FUNCTION_BLOCK FB_WriteRegsExample
VAR
	fbWriteRegisters : FB_MBWriteRegs;
	nWriteValueArray : ARRAY[0..9] OF INT;
	wWriteRegsValueConvertToWord : WORD;
	eWriteState : (WAIT, TRIGGER, WRITE);
	fbTriggerStart : R_TRIG;
	fbTriggerStop : R_TRIG;
	//cbLength: UINT;
	
END_VAR

fbTriggerStart();
IF fbTriggerStart.Q THEN
	IF eWriteState = WAIT THEN
		 eWriteState := TRIGGER;
	END_IF
END_IF
IF fbTriggerStop.CLK THEN
	fbWriteRegisters(bExecute := FALSE);
	eWriteState := WAIT;
END_IF
CASE eWriteState OF
	WAIT : 
	// NOTHING
	TRIGGER : 
	 //wWriteRegsValueConvertToWord := TO_WORD(nWriteValueInt);
	 (*fbWriteRegisters(
		sIPAddr:= '192.168.10.1', 
		nTCPPort:= 502, 
		nUnitID:= 16#FF, 
		nMBAddr:= 0, 
		nValue:= wWriteRegsValueConvertToWord, 
		bExecute:= TRUE, 
		tTimeout:= , 
		bBusy=> , 
		bError=> , 
		nErrId=> ); *)
	fbWriteRegisters(
		sIPAddr:= '192.168.10.1', 
		nTCPPort:= 502, 
		nUnitID:= 16#FF, 
		nQuantity:= 10, 
		nMBAddr:= 0, 
		cbLength:= SIZEOF(nWriteValueArray), 
		pSrcAddr:= ADR(nWriteValueArray), 
		bExecute:= TRUE, 
		tTimeout:= , 
		bBusy=> , 
		bError=> , 
		nErrId=> );
	eWriteState := WRITE;
	WRITE :
	fbWriteRegisters(bExecute := FALSE);
	IF NOT fbWriteRegisters.bBusy AND NOT fbWriteRegisters.bError AND NOT fbTriggerStop.CLK  THEN 
				 eWriteState := TRIGGER;
	ELSIF fbWriteRegisters.bError  THEN
 			eWriteState := WAIT;
		
	END_IF
		
END_CASE

END_FUNCTION_BLOCK

(* stored: Version 1.1.0.1, ProductVersion 3.1.4024.16
   POU FB_WriteRegsExample: Id {d5d57119-5488-416e-878a-e77aa9c88dfa}, SpecialFunc None *)
